(* PLC project CoDeSys External Library Template, WAGO e!COCKPIT e!COCKPIT, author 3S - Smart Software Solutions GmbH *)
(* stored: creationDateTime 2019-10-29T12:37:19.3459586, version 3.5.5.30, modificationDateTime 2019-10-29T12:36:39.3744516, organization 3S - Smart Software Solutions GmbH *)
(* Library project template with all possible element types, docu and a sample project structure *)

(* Autor: Paweł Kąkol, 2018-09-03-PK Prawa majątkowe: Solwena Sp. z o.o., Aktualizacje: 2019-02-18-AWy: alarm czujnika temperatury 2019-02-18-AWy: zmiana klas alarmów Opis: enum służy do definicji klas alarmów w fb węzła Climatix POL63x na budynkach PPP Sopot (ENGIE) *)
{attribute 'qualified_only'}
{attribute 'strict'}
TYPE enumPPPSDestratyfikatorTBOXErrorKlasa : (BrakKomunikacji := enumKlasaAlarmu.AwariaAutomatyki, AlarmCzujnika := enumKlasaAlarmu.AwariaAutomatyki);
END_TYPE
